{attribute 'qualified_only'}
VAR_GLOBAL
    nTooLow : UDINT;
    nTooHigh : UDINT;
    nDivByZero : UDINT;
END_VAR

(* stored: Version 1.1.0.1, ProductVersion 3.1.4022.18
   GVL GVL_CheckBounds: Id {3372cf4f-1868-41ef-b254-996be3d92c90} *)
